// TIA Portal V20 export
// export: Created 2026-08-23T16:24:52.4288924Z, ExportSetting WithDefaults, DisplayName Totally Integrated Automation Portal, DisplayVersion V20 Update 5, DisplayName TIA Portal Openness, DisplayVersion V20 Update 4, DisplayName TIA Portal Version Control Interface, DisplayVersion V20 Update 5, DisplayName SINAMICS Startdrive Advanced, DisplayVersion V20, DisplayName SINAMICS DCC, DisplayVersion V20, DisplayName SINAMICS Startdrive G130, G150, S120, S150, SINAMICS MV, G220, S200, S210, DisplayVersion V20, DisplayName SINAMICS Startdrive G110M, G120, G120C, G120D, G120P, G115D, DisplayVersion V20, DisplayName STEP 7 Professional, DisplayVersion V20 Update 5, DisplayName STEP 7 Safety, DisplayVersion V20 Update 2, DisplayName WinCC Basic/Comfort/Advanced, DisplayVersion V20 Update 5, DisplayName WinCC Unified, DisplayVersion V20 Update 5
ORGANIZATION_BLOCK "Main"   // OB1, LAD, ProgramCycle
TITLE = "Main Program Sweep (Cycle)"
{ S7_Optimized_Access := 'TRUE' }
VERSION : 0.1
// stored: AutoNumber true, IsIECCheckEnabled false, SetENOAutomatically false
   VAR_INPUT
      Initial_Call : Bool;   // Initial call of this OB
      Remanence : Bool;   // =True, if remanent data are available
   END_VAR
BEGIN

REGION Network 1: Hopper-Blockage Stimulus Model
   // Advances the commanded timeline the hopper-blockage monitor is tested against and presents it to the input buffer's test members. It runs ahead of the input map because for a commanded input the model is the field: the map that follows chooses between the terminal and the test member, and it must find this scan's commanded state rather than the previous scan's. Outside a run it drives nothing and the map reads the field.
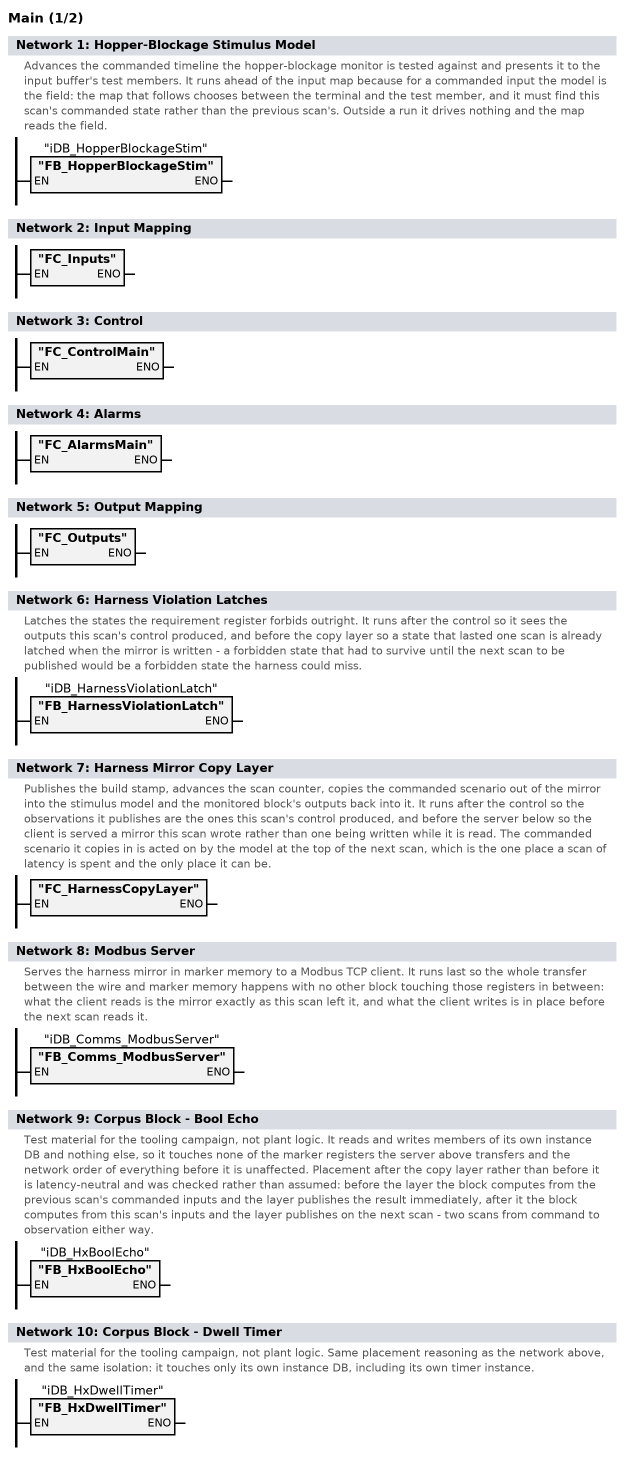
   RUNG wire#powerrail
      "iDB_HopperBlockageStim"()
   END_RUNG
   // the same network as SCL:
   "iDB_HopperBlockageStim"();   // "FB_HopperBlockageStim"
END_REGION

REGION Network 2: Input Mapping
   RUNG wire#powerrail
      "FC_Inputs"()
   END_RUNG
   // the same network as SCL:
   "FC_Inputs"();
END_REGION

REGION Network 3: Control
   RUNG wire#powerrail
      "FC_ControlMain"()
   END_RUNG
   // the same network as SCL:
   "FC_ControlMain"();
END_REGION

REGION Network 4: Alarms
   RUNG wire#powerrail
      "FC_AlarmsMain"()
   END_RUNG
   // the same network as SCL:
   "FC_AlarmsMain"();
END_REGION

REGION Network 5: Output Mapping
   RUNG wire#powerrail
      "FC_Outputs"()
   END_RUNG
   // the same network as SCL:
   "FC_Outputs"();
END_REGION

REGION Network 6: Harness Violation Latches
   // Latches the states the requirement register forbids outright. It runs after the control so it sees the outputs this scan's control produced, and before the copy layer so a state that lasted one scan is already latched when the mirror is written - a forbidden state that had to survive until the next scan to be published would be a forbidden state the harness could miss.
   RUNG wire#powerrail
      "iDB_HarnessViolationLatch"()
   END_RUNG
   // the same network as SCL:
   "iDB_HarnessViolationLatch"();   // "FB_HarnessViolationLatch"
END_REGION

REGION Network 7: Harness Mirror Copy Layer
   // Publishes the build stamp, advances the scan counter, copies the commanded scenario out of the mirror into the stimulus model and the monitored block's outputs back into it. It runs after the control so the observations it publishes are the ones this scan's control produced, and before the server below so the client is served a mirror this scan wrote rather than one being written while it is read. The commanded scenario it copies in is acted on by the model at the top of the next scan, which is the one place a scan of latency is spent and the only place it can be.
   RUNG wire#powerrail
      "FC_HarnessCopyLayer"()
   END_RUNG
   // the same network as SCL:
   "FC_HarnessCopyLayer"();
END_REGION

REGION Network 8: Modbus Server
   // Serves the harness mirror in marker memory to a Modbus TCP client. It runs last so the whole transfer between the wire and marker memory happens with no other block touching those registers in between: what the client reads is the mirror exactly as this scan left it, and what the client writes is in place before the next scan reads it.
   RUNG wire#powerrail
      "iDB_Comms_ModbusServer"()
   END_RUNG
   // the same network as SCL:
   "iDB_Comms_ModbusServer"();   // "FB_Comms_ModbusServer"
END_REGION

REGION Network 9: Corpus Block - Bool Echo
   // Test material for the tooling campaign, not plant logic. It reads and writes members of its own instance DB and nothing else, so it touches none of the marker registers the server above transfers and the network order of everything before it is unaffected. Placement after the copy layer rather than before it is latency-neutral and was checked rather than assumed: before the layer the block computes from the previous scan's commanded inputs and the layer publishes the result immediately, after it the block computes from this scan's inputs and the layer publishes on the next scan - two scans from command to observation either way.
   RUNG wire#powerrail
      "iDB_HxBoolEcho"()
   END_RUNG
   // the same network as SCL:
   "iDB_HxBoolEcho"();   // "FB_HxBoolEcho"
END_REGION

REGION Network 10: Corpus Block - Dwell Timer
   // Test material for the tooling campaign, not plant logic. Same placement reasoning as the network above, and the same isolation: it touches only its own instance DB, including its own timer instance.
   RUNG wire#powerrail
      "iDB_HxDwellTimer"()
   END_RUNG
   // the same network as SCL:
   "iDB_HxDwellTimer"();   // "FB_HxDwellTimer"
END_REGION

REGION Network 11: Corpus Block - Int Sum
   // Test material for the tooling campaign, not plant logic. Same placement reasoning as the networks above, and the same isolation: it touches only its own instance DB.
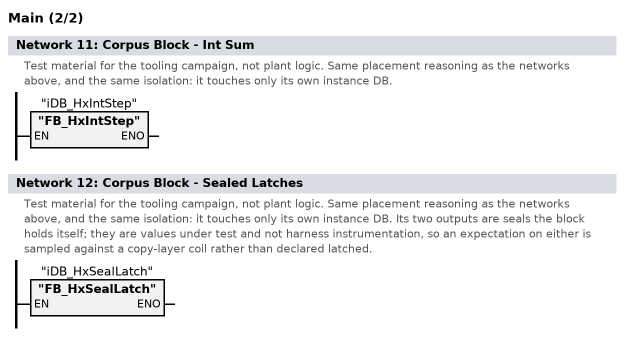
   RUNG wire#powerrail
      "iDB_HxIntStep"()
   END_RUNG
   // the same network as SCL:
   "iDB_HxIntStep"();   // "FB_HxIntStep"
END_REGION

REGION Network 12: Corpus Block - Sealed Latches
   // Test material for the tooling campaign, not plant logic. Same placement reasoning as the networks above, and the same isolation: it touches only its own instance DB. Its two outputs are seals the block holds itself; they are values under test and not harness instrumentation, so an expectation on either is sampled against a copy-layer coil rather than declared latched.
   RUNG wire#powerrail
      "iDB_HxSealLatch"()
   END_RUNG
   // the same network as SCL:
   "iDB_HxSealLatch"();   // "FB_HxSealLatch"
END_REGION
END_ORGANIZATION_BLOCK
